INTERFACE I_SingleDirectionMotor

METHOD Start
VAR_INPUT
END_VAR
END_METHOD

METHOD Stop
VAR_INPUT
END_VAR
END_METHOD

END_INTERFACE

(* stored: Version 1.1.0.1, ProductVersion 3.1.4024.11
   Itf I_SingleDirectionMotor: Id {9238e941-d894-4aa5-b8c5-1d053e31c834}
   Method Start: Id {01beb6f7-92f1-4bb9-b8fc-e4c1aada33a8}
   Method Stop: Id {ee299f31-c451-4c7a-9b02-ee1c094ca48e} *)
